TYPE ST_FlowScale :
STRUCT
	fMaxFlowInput : LREAL; 
	fMinFlowInput : LREAL;
    fNeutralFlowInput : LREAL; 
	fNeutralDeadband : LREAL; 
	fMaxFlowOutput : LREAL; 
	fMinFlowOutput : LREAL; 
	fNeutralFlowOutput : LREAL; 
END_STRUCT
END_TYPE

(* stored: Version 1.1.0.1, ProductVersion 3.1.4024.12
   DUT ST_FlowScale: Id {a3bb7253-5222-4430-ba6e-2bba1e88bd05} *)
